(* IEC 61131-3 sources: IRIS-Project/LASAL CONTROL SOFTWARE/LasalProject_2025_09_12/Class/EStopManager, 1 file *)

(* ---- EStopManager.st ---- *)
(*!
<Class
	Name               = "EStopManager"
	Revision           = "0.0"
	RealtimeTask       = "true"
	DefRealtime        = "50 ms"
	CyclicTask         = "false"
	BackgroundTask     = "false"
	Sigmatek           = "false"
	OSInterface        = "false"
	HighPriority       = "false"
	Automatic          = "false"
	UpdateMode         = "Prescan"
	SharedCommandTable = "true"
	Objectsize         = "(420,1080)">
	<Channels>
		<Server Name="ClassSvr" Visualized="false" Initialize="false" WriteProtected="true" Retentive="false"/>
		<Server Name="E_Signal" Visualized="false" Initialize="false" WriteProtected="true" Retentive="false"/>
		<Client Name="Client" Required="true" Internal="false"/>
		<Client Name="M1_EN1" Required="true" Internal="false"/>
		<Client Name="M1_EN2" Required="true" Internal="false"/>
		<Client Name="M2_EN1" Required="true" Internal="false"/>
		<Client Name="M2_EN2" Required="true" Internal="false"/>
		<Client Name="M3_EN1" Required="true" Internal="false"/>
		<Client Name="M3_EN2" Required="true" Internal="false"/>
		<Client Name="M4_EN1" Required="true" Internal="false"/>
		<Client Name="M4_EN2" Required="true" Internal="false"/>
		<Client Name="M5_EN1" Required="true" Internal="false"/>
		<Client Name="M5_EN2" Required="true" Internal="false"/>
		<Client Name="M6_EN1" Required="true" Internal="false"/>
		<Client Name="M6_EN2" Required="true" Internal="false"/>
	</Channels>
	<Separators>
		<Clients>
			<SepChn Position="2"/>
			<SepChn Position="5"/>
			<SepChn Position="8"/>
			<SepChn Position="11"/>
			<SepChn Position="14"/>
		</Clients>
	</Separators>
</Class>
*)
EStopManager : CLASS
  //Servers:
	ClassSvr 	: SvrChCmd_DINT;
	E_Signal 	: SvrCh_DINT;
  //Clients:
	M1_EN1 	: CltCh_DINT;
	M1_EN2 	: CltCh_DINT;
	M2_EN1 	: CltCh_DINT;
	M2_EN2 	: CltCh_DINT;
	M3_EN1 	: CltCh_DINT;
	M3_EN2 	: CltCh_DINT;
	M4_EN1 	: CltCh_DINT;
	M4_EN2 	: CltCh_DINT;
	M5_EN1 	: CltCh_DINT;
	M5_EN2 	: CltCh_DINT;
	M6_EN1 	: CltCh_DINT;
	M6_EN2 	: CltCh_DINT;
	Client 	: CltCh_DINT;
  //Variables:
		ArrayEN : ARRAY [0..11] OF DINT;

		v_E_Signal 	: BOOL;
		i 	: DINT;
		Variable 	: DINT;
  //Functions:

	FUNCTION VIRTUAL GLOBAL Init;

	FUNCTION VIRTUAL GLOBAL RtWork
		VAR_INPUT
			EAX 	: UDINT;
		END_VAR
		VAR_OUTPUT
			state (EAX) 	: UDINT;
		END_VAR;
  //Tables:
	FUNCTION @STD
		VAR_OUTPUT
			ret_code	: CONFSTATES;
		END_VAR;
	FUNCTION GLOBAL TAB @CT_;
END_CLASS;

FUNCTION VIRTUAL GLOBAL EStopManager::RtWork
	VAR_INPUT
		EAX 	: UDINT;
	END_VAR
	VAR_OUTPUT
		state (EAX) 	: UDINT;
	END_VAR

M1_EN1:=1;

for i:=0 to 11 by 1 do
  ArrayEN[0]  :=  M1_EN1;
  ArrayEN[1]  :=  M1_EN2;
  ArrayEN[2]  :=  M2_EN1.Read();
  ArrayEN[3]  :=  M2_EN2.Read();
  ArrayEN[4]  :=  M3_EN1.Read();
  ArrayEN[5]  :=  M3_EN2.Read();
  ArrayEN[6]  :=  M4_EN1.Read();
  ArrayEN[7]  :=  M4_EN2.Read();
  ArrayEN[8]  :=  M5_EN1.Read();
  ArrayEN[9]  :=  M5_EN2.Read();
  ArrayEN[10] :=  M6_EN1.Read();
  ArrayEN[11] :=  M6_EN2.Read();

end_for;

for i:=0 to 11 by 1 do
  if ArrayEN[i]=0 then
    v_E_Signal:=1;
    E_Signal:=v_E_Signal;
  end_if;

end_for;

	state := READY;

END_FUNCTION

FUNCTION VIRTUAL GLOBAL EStopManager::Init

v_E_Signal:=0;
i:=0;

END_FUNCTION
